// TIA Portal project "Project4" (V15.1)

(* hardware
DEVICE "S7300/ET200M station_1"  S7-300 station
   slot 0: "Rail_0"  Rail  6ES7 390-1***0-0AA0
   slot 2: "PLC_1"  CPU 312  6ES7 312-1AE14-0AB0  V3.3
      slot 0: "MPI interface_1"  MPI
*)

// ===== PLC "PLC_1"  CPU 312 =====

VAR_GLOBAL   // PLC tag table "Default tag table"
   "LAH_in" AT %I0.0 : Bool;
   "LAL_in" AT %I0.1 : Bool;
   "Uklj_kon_1_out" AT %Q4.0 : Bool;
   "Uklj_kon_2_out" AT %Q4.1 : Bool;
   "Rucni rezim rada" AT %M0.0 : Bool;
   "Automatski rezim rada" AT %M0.1 : Bool;
   "Tag_1" AT %M1.0 : Bool;
   "Tag_2" AT %M1.1 : Bool;
   "Tag_3" AT %M0.2 : Bool;
END_VAR

DATA_BLOCK "Data_block_1"   // DB10
{ S7_Optimized_Access := 'FALSE' }
VERSION : 0.1
   VAR
      Start_1 : Bool;
      Stop_1 : Bool;
      Start_2 : Bool;
      Stop_2 : Bool;
      Auto_man : Bool;
   END_VAR
BEGIN
END_DATA_BLOCK

FUNCTION "Block_1" : Void   // FC1, LAD
{ S7_Optimized_Access := 'FALSE' }
VERSION : 0.1
BEGIN

REGION Network 1: Rezim rada
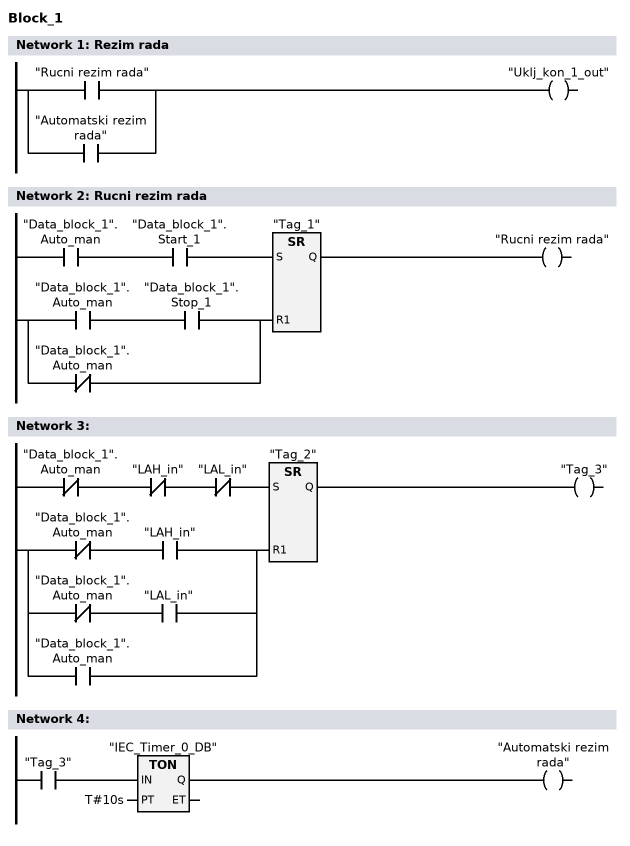
   RUNG wire#powerrail
      Contact( "Rucni rezim rada" )
      wire#w1
      Coil( "Uklj_kon_1_out" )
   END_RUNG
   RUNG wire#powerrail
      Contact( "Automatski rezim rada" )
   END_RUNG wire#w1
   // the same network as SCL:
   "Uklj_kon_1_out" := "Rucni rezim rada" OR "Automatski rezim rada";
END_REGION

REGION Network 2: Rucni rezim rada
   RUNG wire#powerrail
      Contact( "Data_block_1".Auto_man )
      Contact( "Data_block_1".Start_1 )
      S_SR(operand := "Tag_1", r1 := wire#w1)
      Coil( "Rucni rezim rada" )
   END_RUNG
   RUNG wire#powerrail
      Contact( "Data_block_1".Auto_man )
      Contact( "Data_block_1".Stop_1 )
   END_RUNG wire#w1
   RUNG wire#powerrail
      I_Contact( "Data_block_1".Auto_man )
   END_RUNG wire#w1
   // the same network as SCL:
   IF "Data_block_1".Auto_man AND "Data_block_1".Start_1 THEN
       "Tag_1" := TRUE;   // SR flip-flop
   END_IF;
   IF ("Data_block_1".Auto_man AND "Data_block_1".Stop_1) OR NOT "Data_block_1".Auto_man THEN
       "Tag_1" := FALSE;
   END_IF;
   "Rucni rezim rada" := "Tag_1";
END_REGION

REGION Network 3
   RUNG wire#powerrail
      I_Contact( "Data_block_1".Auto_man )
      I_Contact( "LAH_in" )
      I_Contact( "LAL_in" )
      S_SR(operand := "Tag_2", r1 := wire#w1)
      Coil( "Tag_3" )
   END_RUNG
   RUNG wire#powerrail
      I_Contact( "Data_block_1".Auto_man )
      Contact( "LAH_in" )
   END_RUNG wire#w1
   RUNG wire#powerrail
      I_Contact( "Data_block_1".Auto_man )
      Contact( "LAL_in" )
   END_RUNG wire#w1
   RUNG wire#powerrail
      Contact( "Data_block_1".Auto_man )
   END_RUNG wire#w1
   // the same network as SCL:
   IF NOT "Data_block_1".Auto_man AND NOT "LAH_in" AND NOT "LAL_in" THEN
       "Tag_2" := TRUE;   // SR flip-flop
   END_IF;
   IF (NOT "Data_block_1".Auto_man AND "LAH_in") OR (NOT "Data_block_1".Auto_man AND "LAL_in") OR "Data_block_1".Auto_man THEN
       "Tag_2" := FALSE;
   END_IF;
   "Tag_3" := "Tag_2";
END_REGION

REGION Network 4
   "IEC_Timer_0_DB".TON(IN := "Tag_3", PT := T#10s);
   "Automatski rezim rada" := "IEC_Timer_0_DB".Q;
END_REGION
END_FUNCTION

ORGANIZATION_BLOCK "Main"   // OB1, LAD
TITLE = "Main Program Sweep (Cycle)"
{ S7_Optimized_Access := 'FALSE' }
VERSION : 0.1
   VAR_TEMP
      OB1_EV_CLASS : Byte;   // Bits 0-3 = 1 (Coming event), Bits 4-7 = 1 (Event class 1)
      OB1_SCAN_1 : Byte;   // 1 (Cold restart scan 1 of OB 1), 3 (Scan 2-n of OB 1)
      OB1_PRIORITY : Byte;   // Priority of OB Execution
      OB1_OB_NUMBR : Byte;   // 1 (Organization block 1, OB1)
      OB1_RESERVED_1 : Byte;   // Reserved for system
      OB1_RESERVED_2 : Byte;   // Reserved for system
      OB1_PREV_CYCLE : Int;   // Cycle time of previous OB1 scan (milliseconds)
      OB1_MIN_CYCLE : Int;   // Minimum cycle time of OB1 (milliseconds)
      OB1_MAX_CYCLE : Int;   // Maximum cycle time of OB1 (milliseconds)
      OB1_DATE_TIME : Date_And_Time;   // Date and time OB1 started
   END_VAR
BEGIN

REGION Network 1
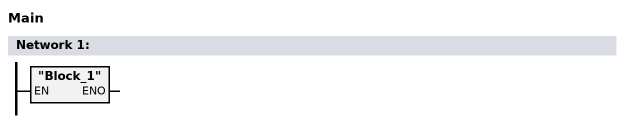
   RUNG wire#powerrail
      "Block_1"()
   END_RUNG
   // the same network as SCL:
   "Block_1"();
END_REGION
END_ORGANIZATION_BLOCK